Staubli VAL3: JogPositve.pgx

public program JogPositve(num x_nAxis, num x_nKey)
begin
  call StepMove(x_nAxis,x_nKey,true)
end
